FUNCTION_BLOCK FB_CCS_SIM
VAR_INPUT
	refTimeObj  : REFERENCE TO FB_TIME; 
END_VAR
VAR_OUTPUT
END_VAR
VAR
	{attribute 'OPC.UA.DA' := '1'}
	cfg:				T_CCS_CFG;
	{attribute 'OPC.UA.DA' := '1'}
	ctrl:				T_CCS_CTRL;
	{attribute 'OPC.UA.DA' := '1'}
	stat:				T_CCS_STAT;
	
    // Tracking data structure are defined in C++ module
	{attribute 'OPC.UA.DA' := '0'}
	i_trk_data          AT %I*: PointingKernelPositions;
	
	{attribute 'OPC.UA.DA' := '0'}
	q_ccs_data          AT %Q*: CcsData;
	
	{attribute 'OPC.UA.DA' := '0'}
	q_mean_coordinates  AT %Q*: TrkMeanCoordinates;
	
	{attribute 'OPC.UA.DA' := '0'}
	q_mudpi_cfg  AT %Q*: T_MUDPI_CFG;
	
END_VAR


// Get parameters
GetParams();

// Set parameters
SetParams();

METHOD FB_init : BOOL
VAR_INPUT
	bInitRetains : BOOL; // if TRUE, the retain variables are initialized (warm start / cold start)
	bInCopyCode : BOOL;  // if TRUE, the instance afterwards gets moved into the copy code (online change)
END_VAR

cfg.site.height              := GVL_TrkSiteConstants.C_HEIGHT;
cfg.site.latitude            := GVL_TrkSiteConstants.C_LATITUDE;
cfg.site.longitude           := GVL_TrkSiteConstants.C_LONGITUDE;
cfg.mudpi.enabled 			 := FALSE;
cfg.mudpi.destination_port	 := 10000;
cfg.mudpi.source_port		 := 8000;
cfg.mudpi.address			 := 0;
cfg.mudpi.component_id	     := 500;
cfg.mudpi.topic_id			 := 10;
ctrl.environment.humidity    := GVL_TrkDefaultEnvironment.C_HUMIDITY;
ctrl.environment.lapserate   := GVL_TrkDefaultEnvironment.C_LAPSERATE;
ctrl.environment.pressure    := GVL_TrkDefaultEnvironment.C_PRESSURE;
ctrl.environment.temperature := GVL_TrkDefaultEnvironment.C_TEMPERATURE;
ctrl.meanCoordinates.alpha   := 0;
ctrl.meanCoordinates.delta   := -890000.0;
ctrl.meanCoordinates.equinox := 2000.0;
END_METHOD

METHOD GetParams
VAR_INPUT
END_VAR

// Assign output variables according input configuration and control.
memcpy(ADR(q_ccs_data.site), ADR(cfg.site), SIZEOF(q_ccs_data.site));	
memcpy(ADR(q_mudpi_cfg), ADR(cfg.mudpi), SIZEOF(q_mudpi_cfg));	
memcpy(ADR(q_ccs_data.environment), ADR(ctrl.environment), SIZEOF(q_ccs_data.environment));
memcpy(ADR(q_mean_coordinates), ADR(ctrl.meanCoordinates), SIZEOF(q_mean_coordinates));
q_ccs_data.equinox := ctrl.equinox;
q_ccs_data.dut := ctrl.dut;
q_ccs_data.wavelength := ctrl.wavelength;
q_mudpi_cfg.address := F_IpAddress2Integer(IpAddress := cfg.ip_address);
END_METHOD

{attribute 'TcRpcEnable':='1'}
METHOD RPC_SetCoordinates : BOOL
VAR_INPUT
	in_alpha:	 LREAL := 000000.0;
	in_delta:    LREAL := 000000.0;
	in_equinox:  LREAL := 2000.0;
END_VAR

ctrl.meanCoordinates.alpha := in_alpha;
ctrl.meanCoordinates.delta := in_delta;
ctrl.meanCoordinates.equinox := in_equinox;
END_METHOD

METHOD SetParams
VAR_INPUT
END_VAR

//memcpy(ADR(stat.apparent), ADR(i_trk_data.apparent), SIZEOF(stat.apparent));
//memcpy(ADR(stat.observed), ADR(i_trk_data.observed), SIZEOF(stat.observed));
memcpy(ADR(stat.data), ADR(i_trk_data), SIZEOF(stat.data));
stat.gui_data.alt := RAD_TO_DEG(stat.data.target_observed_altaz[0]);
stat.gui_data.az := RAD_TO_DEG(stat.data.target_observed_altaz[1]);
stat.gui_data.pa := RAD_TO_DEG(stat.data.parallactic_angle);
stat.gui_data.ra := F_Rad2Hms(stat.data.radec_at_altaz_at_requested_xy[0]);
stat.gui_data.dec := F_Rad2Dms(stat.data.radec_at_altaz_at_requested_xy[1]);
stat.gui_data.north_angle := RAD_TO_DEG(stat.data.north_angle);
stat.gui_data.pupil_angle := RAD_TO_DEG(stat.data.pupil_angle);
stat.gui_data.time_tai := DCTIME64_TO_STRING(refTimeObj.MudpiTimeToDc(stat.data.time_tai));
END_METHOD

END_FUNCTION_BLOCK

(* stored: Version 1.1.0.1, ProductVersion 3.1.4024.11
   POU FB_CCS_SIM: Id {9dd5b39c-af33-4f30-9c96-4ec3ce6ec000}, SpecialFunc None
   Method FB_init: Id {51e92a47-c20e-45ff-8c3a-9298e09677aa}
   Method GetParams: Id {d9e0cfc5-d2af-4af8-aeb7-431bdf29e07c}
   Method RPC_SetCoordinates: Id {3c980e30-80bb-4e69-b66d-f171981c9d87}
   Method SetParams: Id {7b9bdd87-06d7-47d1-b67b-dc712daeb0bc} *)
